(* Logix 5000 project; controller R5_CSS vendor 1 type 14 code 74 rev 19.11; software revision 19.01; part 18 of 20 *)
(* tags used below, declared in another part *)
   PID_TCV406 : PID;
   PID_TCV406_TON : TIMER;
   TC110 : TEMP_CONTROL;   // Quench Water Cartridge Heater Bundle Temp
   TC320 : TEMP_CONTROL;   // COALESCER OIL CHAMBER SHELL TEMPERATURE TRANSMITTER CONTROL
   TC321A : TEMP_CONTROL;   // COALESCER OIL CHAMBER TRANSFER PUMP A TEMPERATURE TRANSMITTER
   TC321B : TEMP_CONTROL;   // COALESCER OIL CHAMBER TRANSFER PUMP B TEMPERATURE TRANSMITTER
   TC406 : TEMP_CONTROL;   // PROCESS WATER POST HX TEMPERATURE CONTROL
   TC406_AUTO_ONS1 : BOOL;
   TC406_LockOut : BOOL;
   TC406_MANUAL_ONS1 : BOOL;
   TC409 : TEMP_CONTROL;   // HX COOLING WATER SUPPLY TEMPERATURE CONTROL
   TC410 : TEMP_CONTROL;   // HX COOLING WATER RETURN TEMPERATURE CONTROL
   TMR_FAULT : DINT;
(* MainProgram, continued *)

ROUTINE TC319A_OilProductHeaterBundleTemp   (* ladder *)
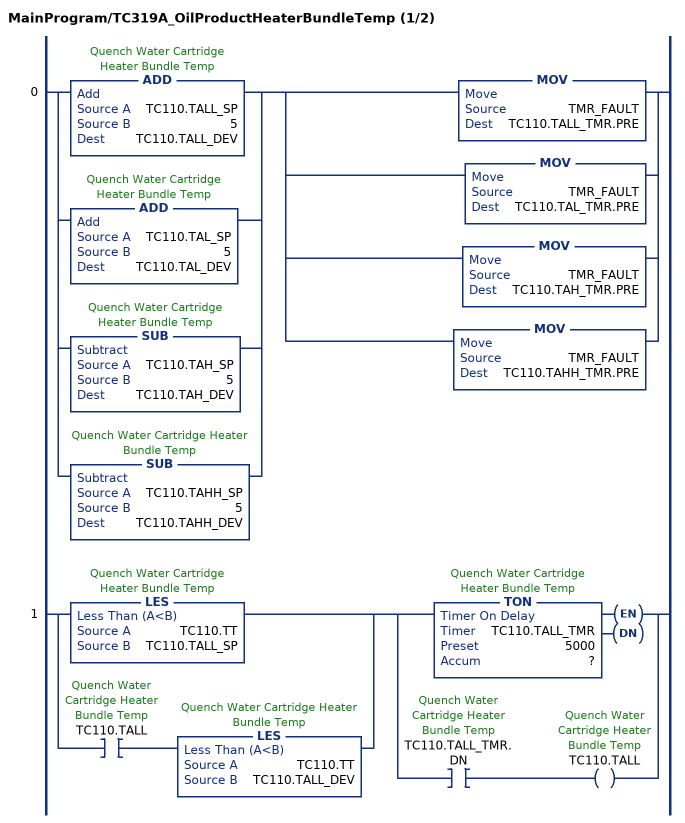
   0: [ADD(TC110.TALL_SP,5,TC110.TALL_DEV) ,ADD(TC110.TAL_SP,5,TC110.TAL_DEV) ,SUB(TC110.TAH_SP,5,TC110.TAH_DEV) ,SUB(TC110.TAHH_SP,5,TC110.TAHH_DEV) ][MOV(TMR_FAULT,TC110.TALL_TMR.PRE) ,MOV(TMR_FAULT,TC110.TAL_TMR.PRE) ,MOV(TMR_FAULT,TC110.TAH_TMR.PRE) ,MOV(TMR_FAULT,TC110.TAHH_TMR.PRE) ];
   1: [LES(TC110.TT,TC110.TALL_SP) ,XIC(TC110.TALL) LES(TC110.TT,TC110.TALL_DEV) ][TON(TC110.TALL_TMR,?,?) ,XIC(TC110.TALL_TMR.DN) OTE(TC110.TALL) ];
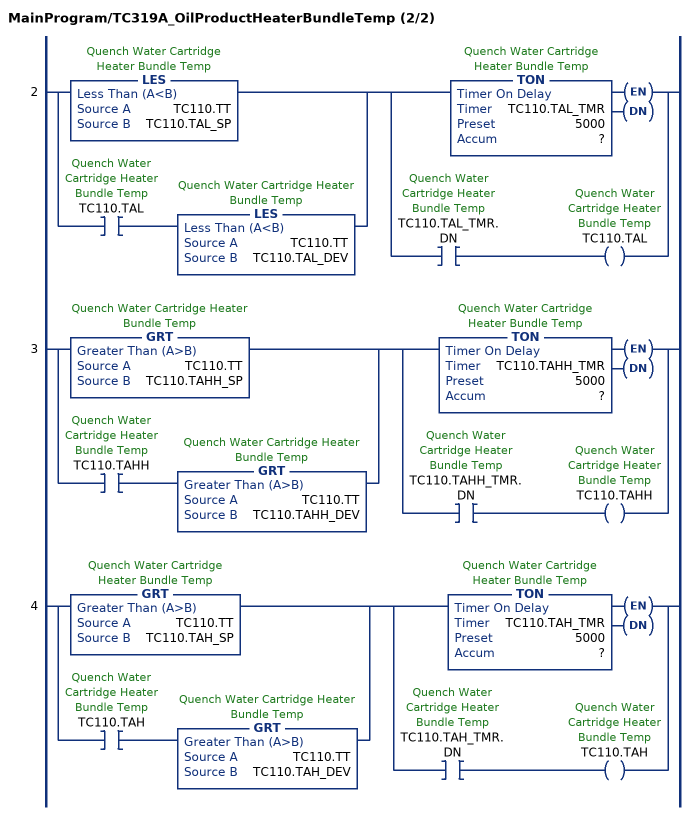
   2: [LES(TC110.TT,TC110.TAL_SP) ,XIC(TC110.TAL) LES(TC110.TT,TC110.TAL_DEV) ][TON(TC110.TAL_TMR,?,?) ,XIC(TC110.TAL_TMR.DN) OTE(TC110.TAL) ];
   3: [GRT(TC110.TT,TC110.TAHH_SP) ,XIC(TC110.TAHH) GRT(TC110.TT,TC110.TAHH_DEV) ][TON(TC110.TAHH_TMR,?,?) ,XIC(TC110.TAHH_TMR.DN) OTE(TC110.TAHH) ];
   4: [GRT(TC110.TT,TC110.TAH_SP) ,XIC(TC110.TAH) GRT(TC110.TT,TC110.TAH_DEV) ][TON(TC110.TAH_TMR,?,?) ,XIC(TC110.TAH_TMR.DN) OTE(TC110.TAH) ];
END_ROUTINE

ROUTINE TC320_OilProductPrePumpTemp   (* ladder *)
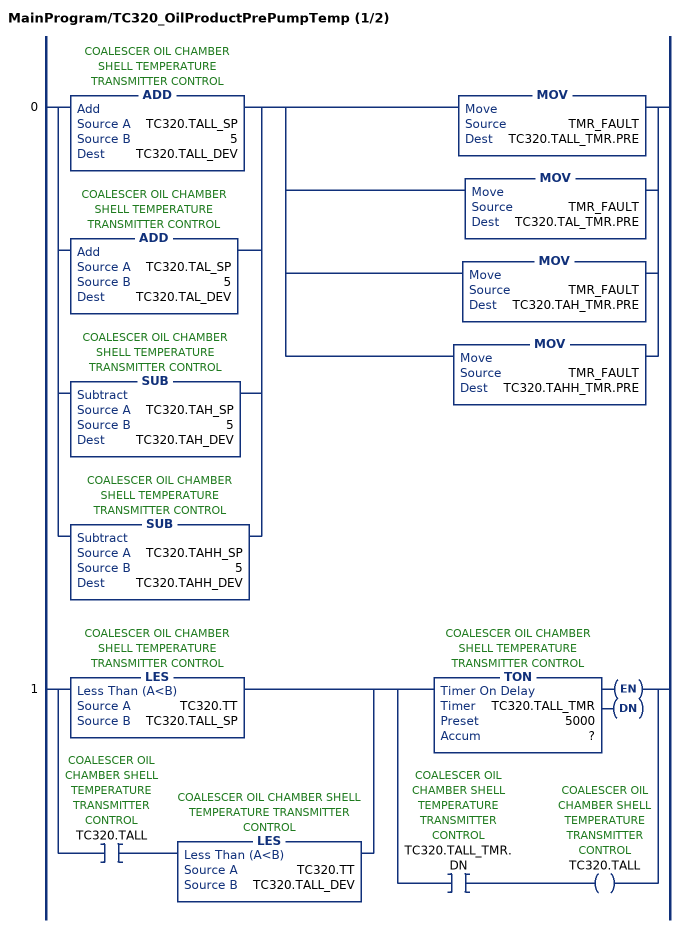
   0: [ADD(TC320.TALL_SP,5,TC320.TALL_DEV) ,ADD(TC320.TAL_SP,5,TC320.TAL_DEV) ,SUB(TC320.TAH_SP,5,TC320.TAH_DEV) ,SUB(TC320.TAHH_SP,5,TC320.TAHH_DEV) ][MOV(TMR_FAULT,TC320.TALL_TMR.PRE) ,MOV(TMR_FAULT,TC320.TAL_TMR.PRE) ,MOV(TMR_FAULT,TC320.TAH_TMR.PRE) ,MOV(TMR_FAULT,TC320.TAHH_TMR.PRE) ];
   1: [LES(TC320.TT,TC320.TALL_SP) ,XIC(TC320.TALL) LES(TC320.TT,TC320.TALL_DEV) ][TON(TC320.TALL_TMR,?,?) ,XIC(TC320.TALL_TMR.DN) OTE(TC320.TALL) ];
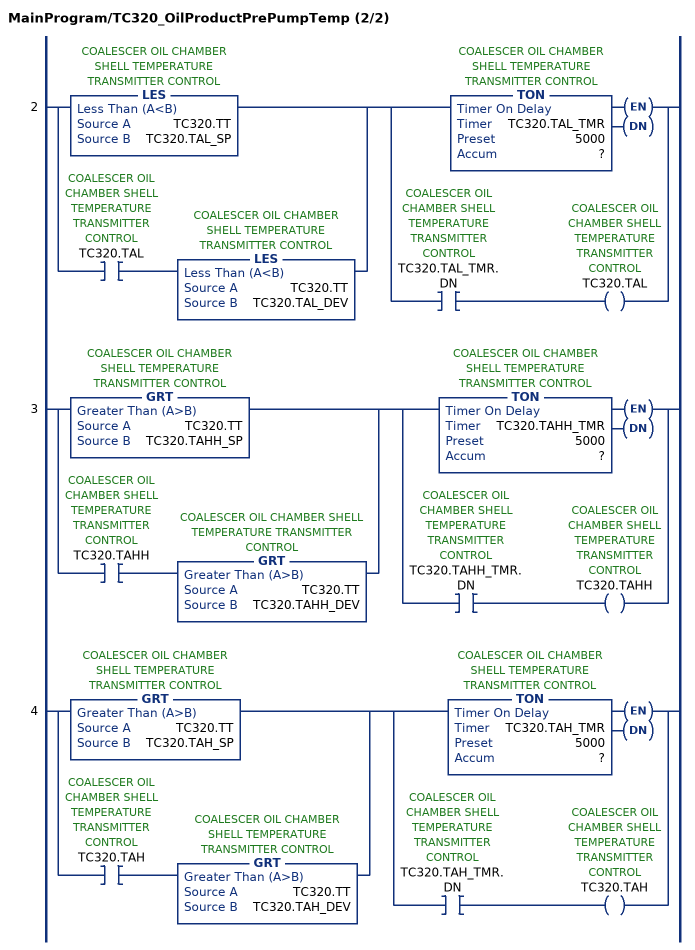
   2: [LES(TC320.TT,TC320.TAL_SP) ,XIC(TC320.TAL) LES(TC320.TT,TC320.TAL_DEV) ][TON(TC320.TAL_TMR,?,?) ,XIC(TC320.TAL_TMR.DN) OTE(TC320.TAL) ];
   3: [GRT(TC320.TT,TC320.TAHH_SP) ,XIC(TC320.TAHH) GRT(TC320.TT,TC320.TAHH_DEV) ][TON(TC320.TAHH_TMR,?,?) ,XIC(TC320.TAHH_TMR.DN) OTE(TC320.TAHH) ];
   4: [GRT(TC320.TT,TC320.TAH_SP) ,XIC(TC320.TAH) GRT(TC320.TT,TC320.TAH_DEV) ][TON(TC320.TAH_TMR,?,?) ,XIC(TC320.TAH_TMR.DN) OTE(TC320.TAH) ];
END_ROUTINE

ROUTINE TC321A_OilProductPumpTemperature   (* ladder *)
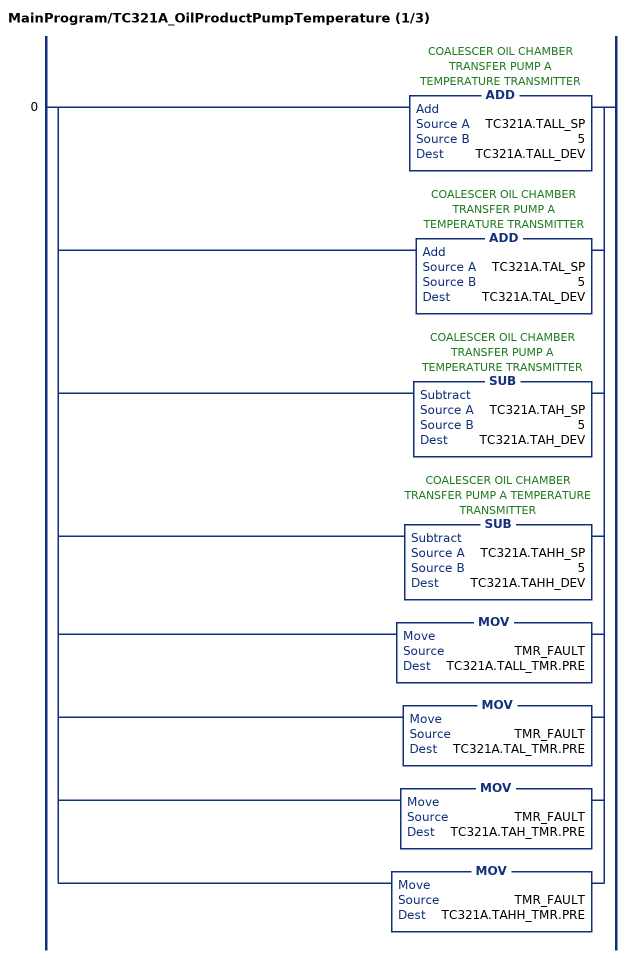
   0: [ADD(TC321A.TALL_SP,5,TC321A.TALL_DEV) ,ADD(TC321A.TAL_SP,5,TC321A.TAL_DEV) ,SUB(TC321A.TAH_SP,5,TC321A.TAH_DEV) ,SUB(TC321A.TAHH_SP,5,TC321A.TAHH_DEV) ,MOV(TMR_FAULT,TC321A.TALL_TMR.PRE) ,MOV(TMR_FAULT,TC321A.TAL_TMR.PRE) ,MOV(TMR_FAULT,TC321A.TAH_TMR.PRE) ,MOV(TMR_FAULT,TC321A.TAHH_TMR.PRE) ];
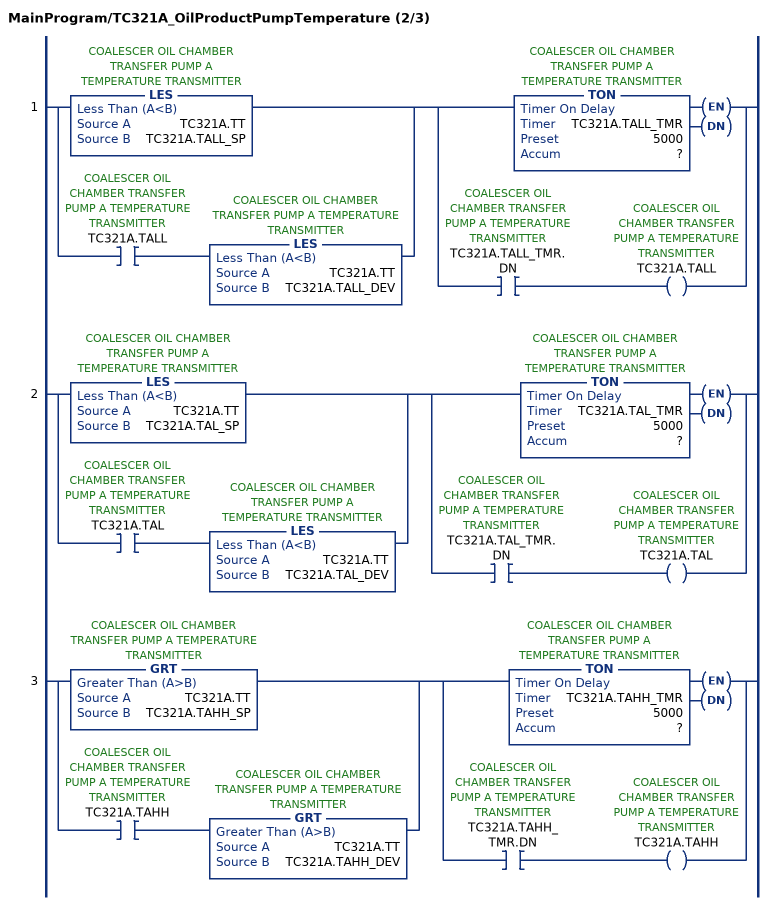
   1: [LES(TC321A.TT,TC321A.TALL_SP) ,XIC(TC321A.TALL) LES(TC321A.TT,TC321A.TALL_DEV) ][TON(TC321A.TALL_TMR,?,?) ,XIC(TC321A.TALL_TMR.DN) OTE(TC321A.TALL) ];
   2: [LES(TC321A.TT,TC321A.TAL_SP) ,XIC(TC321A.TAL) LES(TC321A.TT,TC321A.TAL_DEV) ][TON(TC321A.TAL_TMR,?,?) ,XIC(TC321A.TAL_TMR.DN) OTE(TC321A.TAL) ];
   3: [GRT(TC321A.TT,TC321A.TAHH_SP) ,XIC(TC321A.TAHH) GRT(TC321A.TT,TC321A.TAHH_DEV) ][TON(TC321A.TAHH_TMR,?,?) ,XIC(TC321A.TAHH_TMR.DN) OTE(TC321A.TAHH) ];
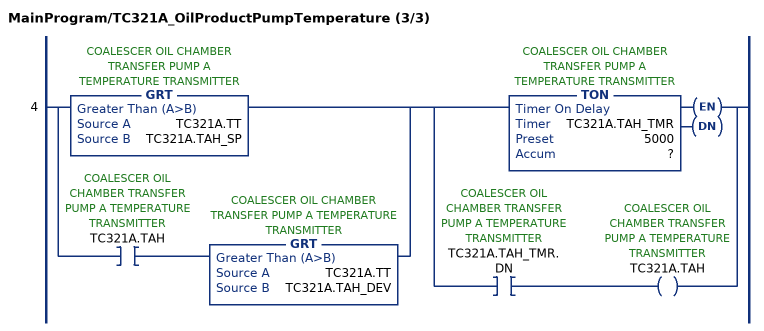
   4: [GRT(TC321A.TT,TC321A.TAH_SP) ,XIC(TC321A.TAH) GRT(TC321A.TT,TC321A.TAH_DEV) ][TON(TC321A.TAH_TMR,?,?) ,XIC(TC321A.TAH_TMR.DN) OTE(TC321A.TAH) ];
END_ROUTINE

ROUTINE TC321B_OilProductPumpTemperature   (* ladder *)
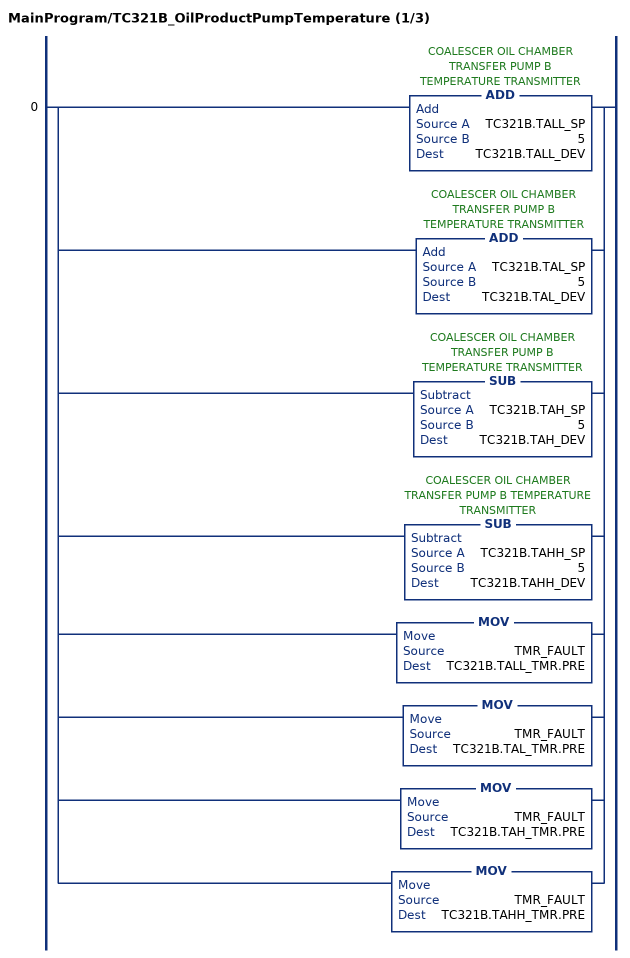
   0: [ADD(TC321B.TALL_SP,5,TC321B.TALL_DEV) ,ADD(TC321B.TAL_SP,5,TC321B.TAL_DEV) ,SUB(TC321B.TAH_SP,5,TC321B.TAH_DEV) ,SUB(TC321B.TAHH_SP,5,TC321B.TAHH_DEV) ,MOV(TMR_FAULT,TC321B.TALL_TMR.PRE) ,MOV(TMR_FAULT,TC321B.TAL_TMR.PRE) ,MOV(TMR_FAULT,TC321B.TAH_TMR.PRE) ,MOV(TMR_FAULT,TC321B.TAHH_TMR.PRE) ];
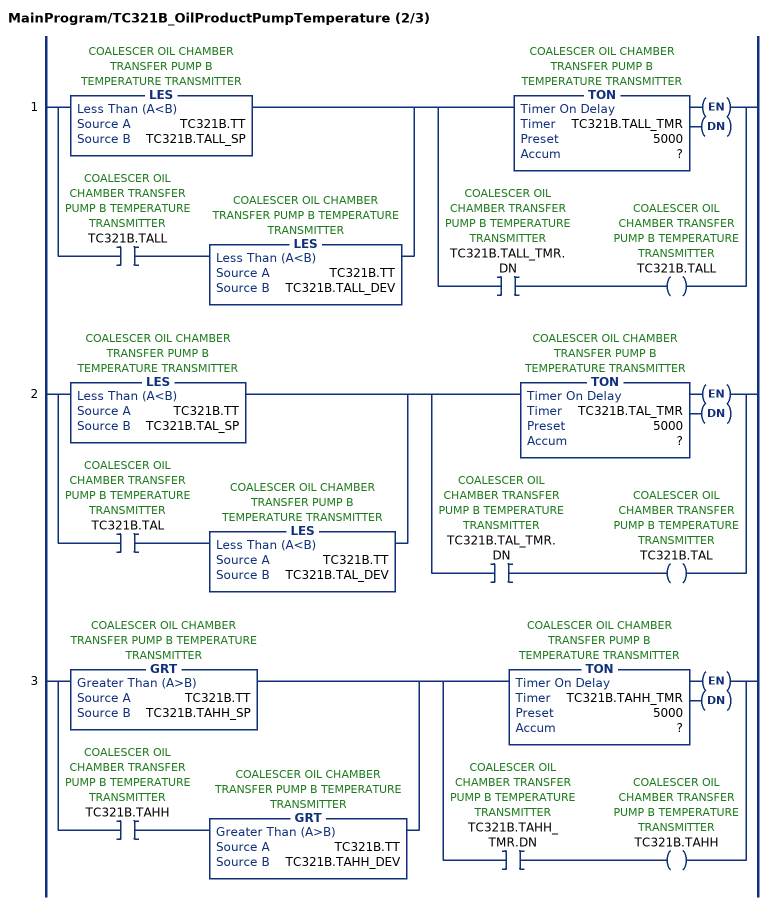
   1: [LES(TC321B.TT,TC321B.TALL_SP) ,XIC(TC321B.TALL) LES(TC321B.TT,TC321B.TALL_DEV) ][TON(TC321B.TALL_TMR,?,?) ,XIC(TC321B.TALL_TMR.DN) OTE(TC321B.TALL) ];
   2: [LES(TC321B.TT,TC321B.TAL_SP) ,XIC(TC321B.TAL) LES(TC321B.TT,TC321B.TAL_DEV) ][TON(TC321B.TAL_TMR,?,?) ,XIC(TC321B.TAL_TMR.DN) OTE(TC321B.TAL) ];
   3: [GRT(TC321B.TT,TC321B.TAHH_SP) ,XIC(TC321B.TAHH) GRT(TC321B.TT,TC321B.TAHH_DEV) ][TON(TC321B.TAHH_TMR,?,?) ,XIC(TC321B.TAHH_TMR.DN) OTE(TC321B.TAHH) ];
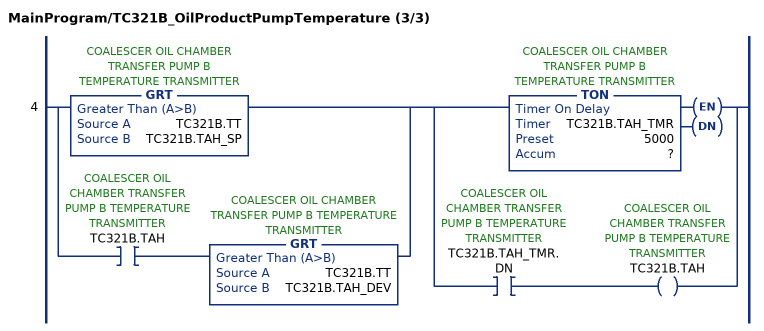
   4: [GRT(TC321B.TT,TC321B.TAH_SP) ,XIC(TC321B.TAH) GRT(TC321B.TT,TC321B.TAH_DEV) ][TON(TC321B.TAH_TMR,?,?) ,XIC(TC321B.TAH_TMR.DN) OTE(TC321B.TAH) ];
END_ROUTINE

ROUTINE TC406_PostHeatExchangeTemp_PID   (* ladder *)
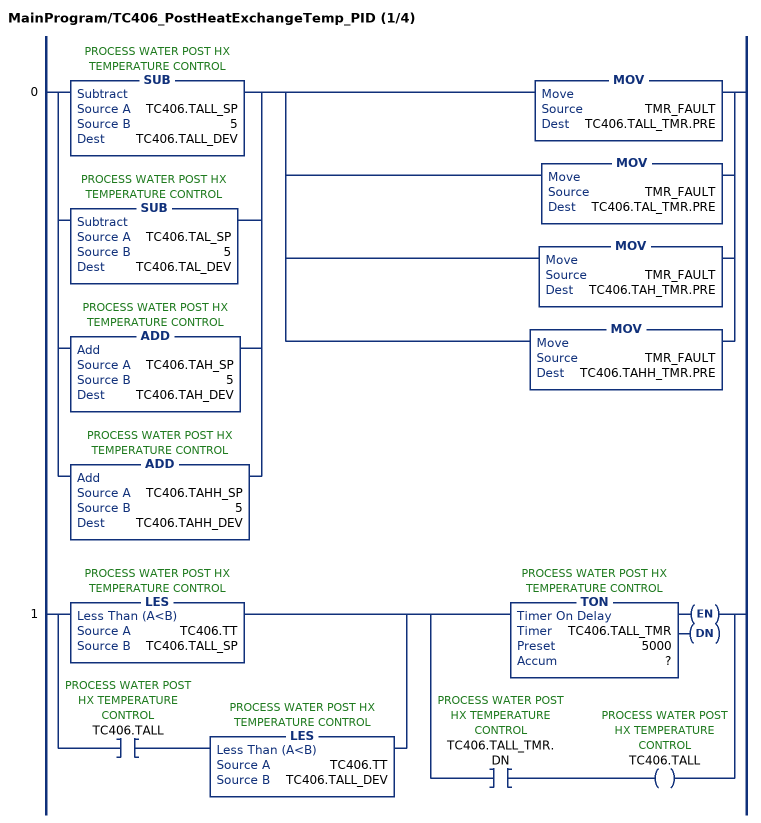
   0: [SUB(TC406.TALL_SP,5,TC406.TALL_DEV) ,SUB(TC406.TAL_SP,5,TC406.TAL_DEV) ,ADD(TC406.TAH_SP,5,TC406.TAH_DEV) ,ADD(TC406.TAHH_SP,5,TC406.TAHH_DEV) ][MOV(TMR_FAULT,TC406.TALL_TMR.PRE) ,MOV(TMR_FAULT,TC406.TAL_TMR.PRE) ,MOV(TMR_FAULT,TC406.TAH_TMR.PRE) ,MOV(TMR_FAULT,TC406.TAHH_TMR.PRE) ];
   1: [LES(TC406.TT,TC406.TALL_SP) ,XIC(TC406.TALL) LES(TC406.TT,TC406.TALL_DEV) ][TON(TC406.TALL_TMR,?,?) ,XIC(TC406.TALL_TMR.DN) OTE(TC406.TALL) ];
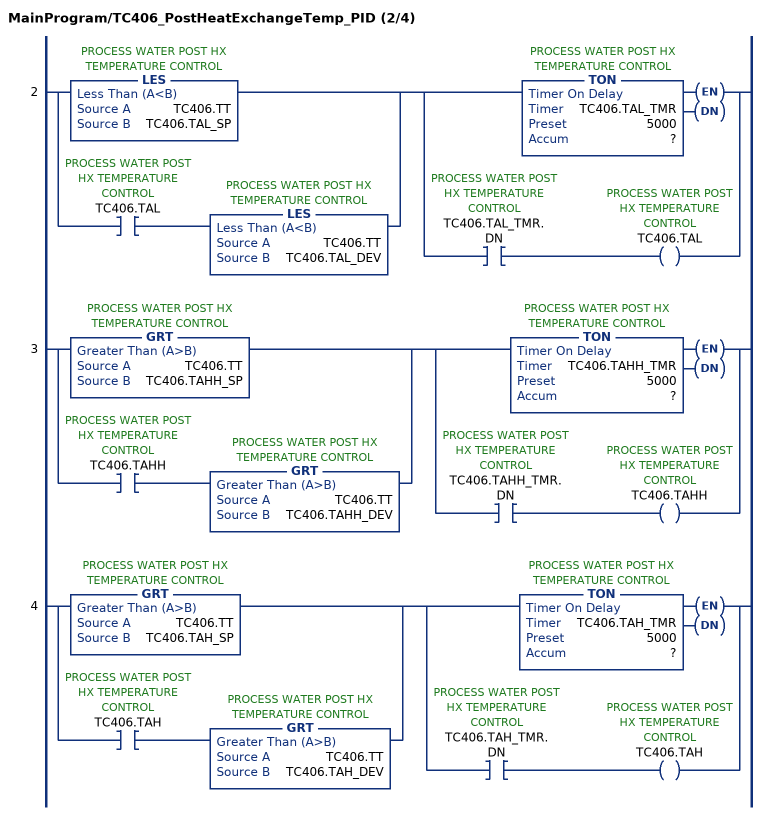
   2: [LES(TC406.TT,TC406.TAL_SP) ,XIC(TC406.TAL) LES(TC406.TT,TC406.TAL_DEV) ][TON(TC406.TAL_TMR,?,?) ,XIC(TC406.TAL_TMR.DN) OTE(TC406.TAL) ];
   3: [GRT(TC406.TT,TC406.TAHH_SP) ,XIC(TC406.TAHH) GRT(TC406.TT,TC406.TAHH_DEV) ][TON(TC406.TAHH_TMR,?,?) ,XIC(TC406.TAHH_TMR.DN) OTE(TC406.TAHH) ];
   4: [GRT(TC406.TT,TC406.TAH_SP) ,XIC(TC406.TAH) GRT(TC406.TT,TC406.TAH_DEV) ][TON(TC406.TAH_TMR,?,?) ,XIC(TC406.TAH_TMR.DN) OTE(TC406.TAH) ];
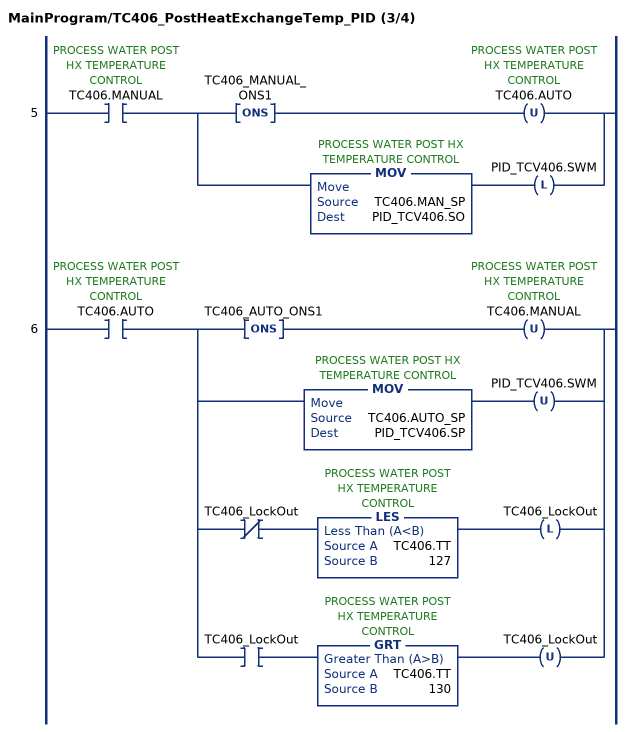
   5: XIC(TC406.MANUAL)[ONS(TC406_MANUAL_ONS1) OTU(TC406.AUTO) ,MOV(TC406.MAN_SP,PID_TCV406.SO) OTL(PID_TCV406.SWM) ];
   6: XIC(TC406.AUTO)[ONS(TC406_AUTO_ONS1) OTU(TC406.MANUAL) ,MOV(TC406.AUTO_SP,PID_TCV406.SP) OTU(PID_TCV406.SWM) ,XIO(TC406_LockOut) LES(TC406.TT,127) OTL(TC406_LockOut) ,XIC(TC406_LockOut) GRT(TC406.TT,130) OTU(TC406_LockOut) ];
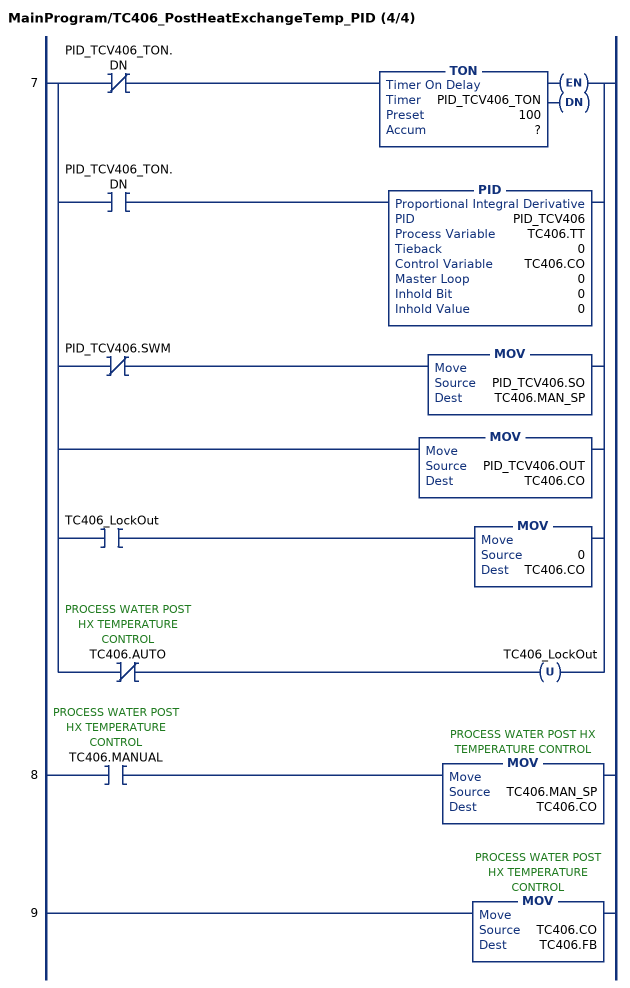
   7: [XIO(PID_TCV406_TON.DN) TON(PID_TCV406_TON,?,?) ,XIC(PID_TCV406_TON.DN) PID(PID_TCV406,TC406.TT,0,TC406.CO,0,0,0) ,XIO(PID_TCV406.SWM) MOV(PID_TCV406.SO,TC406.MAN_SP) ,MOV(PID_TCV406.OUT,TC406.CO) ,XIC(TC406_LockOut) MOV(0,TC406.CO) ,XIO(TC406.AUTO) OTU(TC406_LockOut) ];
   8: XIC(TC406.MANUAL)MOV(TC406.MAN_SP,TC406.CO);
   9: MOV(TC406.CO,TC406.FB);
END_ROUTINE

ROUTINE TC409_PreHeatExchangerCoolTemp   (* ladder *)
// Pre heat exchanger cooling water temperature
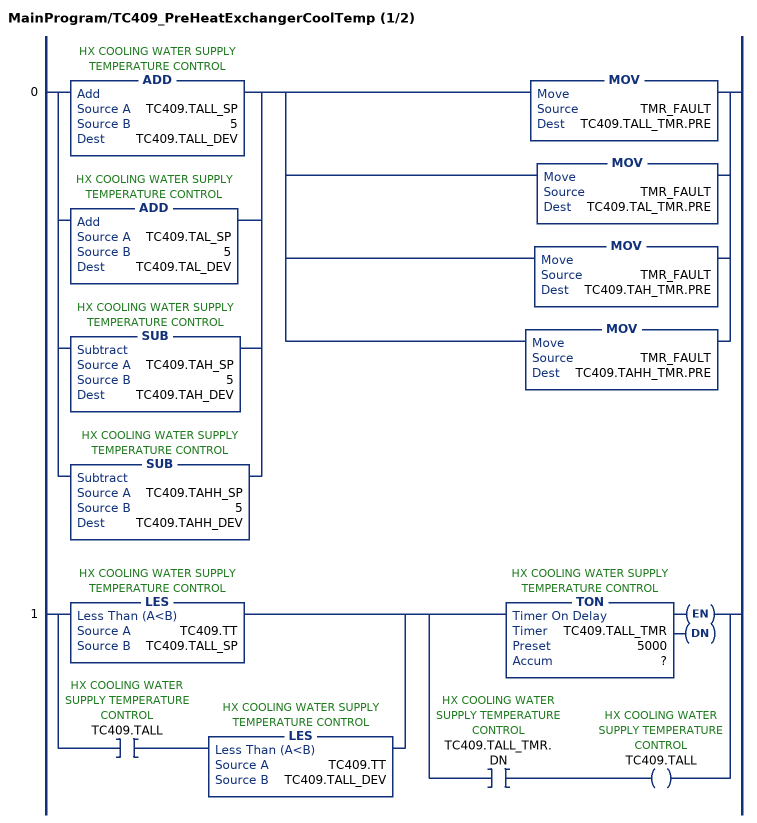
   0: [ADD(TC409.TALL_SP,5,TC409.TALL_DEV) ,ADD(TC409.TAL_SP,5,TC409.TAL_DEV) ,SUB(TC409.TAH_SP,5,TC409.TAH_DEV) ,SUB(TC409.TAHH_SP,5,TC409.TAHH_DEV) ][MOV(TMR_FAULT,TC409.TALL_TMR.PRE) ,MOV(TMR_FAULT,TC409.TAL_TMR.PRE) ,MOV(TMR_FAULT,TC409.TAH_TMR.PRE) ,MOV(TMR_FAULT,TC409.TAHH_TMR.PRE) ];
   1: [LES(TC409.TT,TC409.TALL_SP) ,XIC(TC409.TALL) LES(TC409.TT,TC409.TALL_DEV) ][TON(TC409.TALL_TMR,?,?) ,XIC(TC409.TALL_TMR.DN) OTE(TC409.TALL) ];
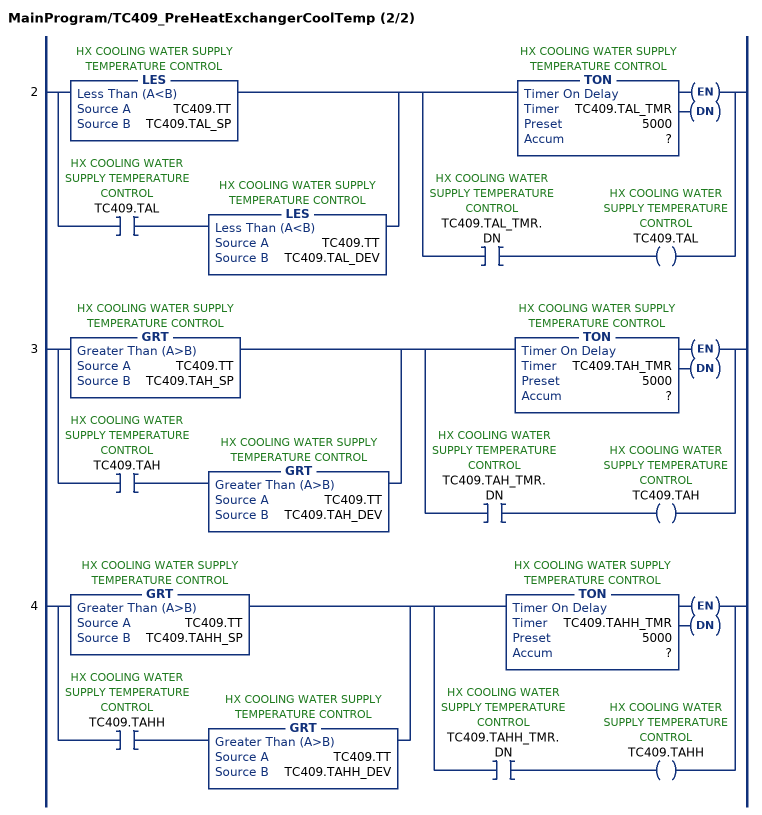
   2: [LES(TC409.TT,TC409.TAL_SP) ,XIC(TC409.TAL) LES(TC409.TT,TC409.TAL_DEV) ][TON(TC409.TAL_TMR,?,?) ,XIC(TC409.TAL_TMR.DN) OTE(TC409.TAL) ];
   3: [GRT(TC409.TT,TC409.TAH_SP) ,XIC(TC409.TAH) GRT(TC409.TT,TC409.TAH_DEV) ][TON(TC409.TAH_TMR,?,?) ,XIC(TC409.TAH_TMR.DN) OTE(TC409.TAH) ];
   4: [GRT(TC409.TT,TC409.TAHH_SP) ,XIC(TC409.TAHH) GRT(TC409.TT,TC409.TAHH_DEV) ][TON(TC409.TAHH_TMR,?,?) ,XIC(TC409.TAHH_TMR.DN) OTE(TC409.TAHH) ];
END_ROUTINE

ROUTINE TC410_PostHeatExchangerCoolTemp   (* ladder *)
// Post heat exchanger cooling water temperature
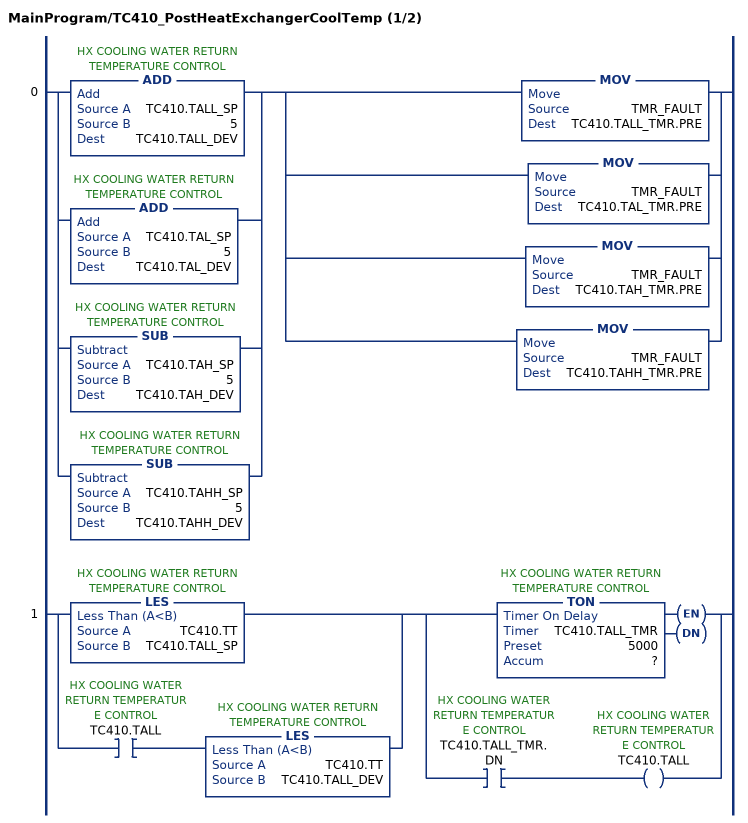
   0: [ADD(TC410.TALL_SP,5,TC410.TALL_DEV) ,ADD(TC410.TAL_SP,5,TC410.TAL_DEV) ,SUB(TC410.TAH_SP,5,TC410.TAH_DEV) ,SUB(TC410.TAHH_SP,5,TC410.TAHH_DEV) ][MOV(TMR_FAULT,TC410.TALL_TMR.PRE) ,MOV(TMR_FAULT,TC410.TAL_TMR.PRE) ,MOV(TMR_FAULT,TC410.TAH_TMR.PRE) ,MOV(TMR_FAULT,TC410.TAHH_TMR.PRE) ];
   1: [LES(TC410.TT,TC410.TALL_SP) ,XIC(TC410.TALL) LES(TC410.TT,TC410.TALL_DEV) ][TON(TC410.TALL_TMR,?,?) ,XIC(TC410.TALL_TMR.DN) OTE(TC410.TALL) ];
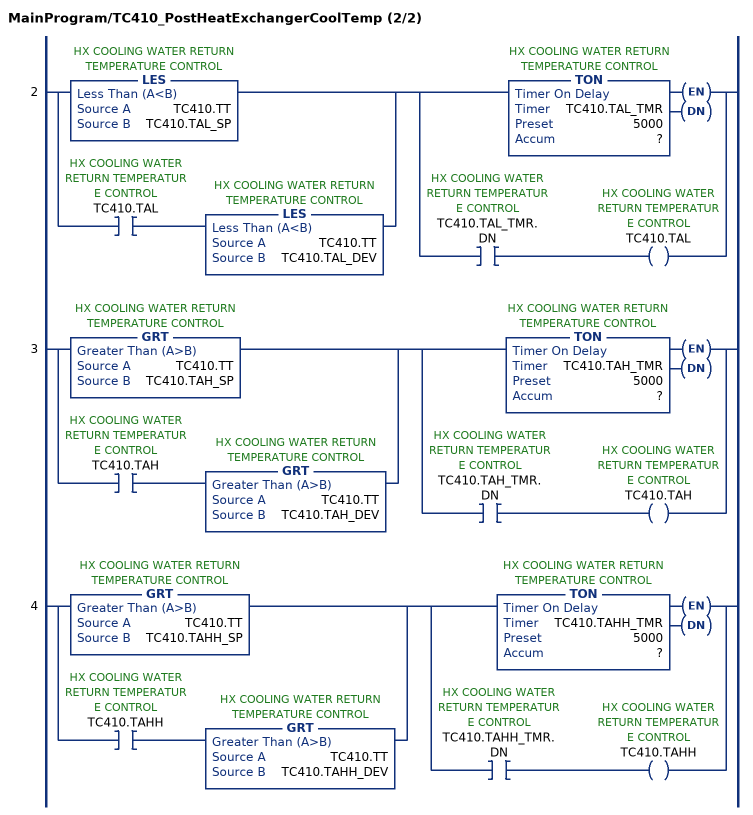
   2: [LES(TC410.TT,TC410.TAL_SP) ,XIC(TC410.TAL) LES(TC410.TT,TC410.TAL_DEV) ][TON(TC410.TAL_TMR,?,?) ,XIC(TC410.TAL_TMR.DN) OTE(TC410.TAL) ];
   3: [GRT(TC410.TT,TC410.TAH_SP) ,XIC(TC410.TAH) GRT(TC410.TT,TC410.TAH_DEV) ][TON(TC410.TAH_TMR,?,?) ,XIC(TC410.TAH_TMR.DN) OTE(TC410.TAH) ];
   4: [GRT(TC410.TT,TC410.TAHH_SP) ,XIC(TC410.TAHH) GRT(TC410.TT,TC410.TAHH_DEV) ][TON(TC410.TAHH_TMR,?,?) ,XIC(TC410.TAHH_TMR.DN) OTE(TC410.TAHH) ];
END_ROUTINE
